PROGRAM pouStationUnits
VAR
	row1: FB_HMI_Control;
	row2: FB_HMI_Control;
	row3: FB_HMI_Control;
	row4: FB_HMI_Control;
	row5: FB_HMI_Control;
	row6: FB_HMI_Control;
	row7: FB_HMI_Control;
	row8: FB_HMI_Control;
	row9: FB_HMI_Control;
	row10: FB_HMI_Control;
	tNumberOfPages: REAL;
	tCalcNumberOfPages: REAL;
	row11: FB_HMI_Control;
	row12: FB_HMI_Control;
	row13: FB_HMI_Control;
	row14: FB_HMI_Control;
	row15: FB_HMI_Control;
	row16: FB_HMI_Control;
	row17: FB_HMI_Control;
	row18: FB_HMI_Control;
	row19: FB_HMI_Control;
	row20: FB_HMI_Control;
	row21: FB_HMI_Control;
	row22: FB_HMI_Control;
	row23: FB_HMI_Control;
	row24: FB_HMI_Control;
	//StationNativeMotionRows: ARRAY[0..99] OF typeMotionRow;
	ceil: LREAL;
END_VAR

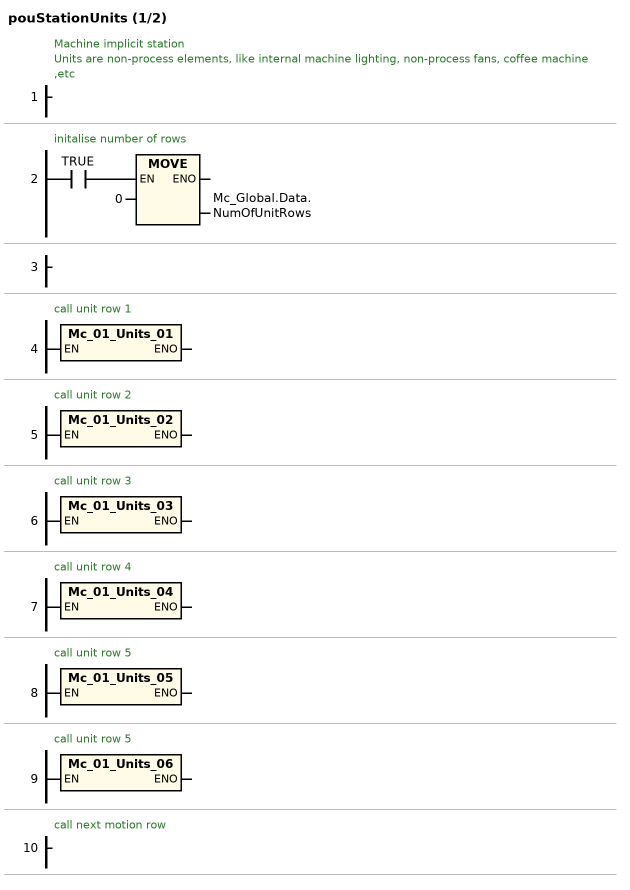
// NETWORK 1
// Machine implicit station
// Units are non-process elements, like internal machine lighting, non-process fans, coffee machine ,etc

// NETWORK 2
// initalise number of rows
Mc_Global.Data.NumOfUnitRows := 0;

// NETWORK 3

// NETWORK 4
// call unit row 1
Mc_01_Units_01();

// NETWORK 5
// call unit row 2
Mc_01_Units_02();

// NETWORK 6
// call unit row 3
Mc_01_Units_03();

// NETWORK 7
// call unit row 4
Mc_01_Units_04();

// NETWORK 8
// call unit row 5
Mc_01_Units_05();

// NETWORK 9
// call unit row 5
Mc_01_Units_06();

// NETWORK 10
// call next motion row

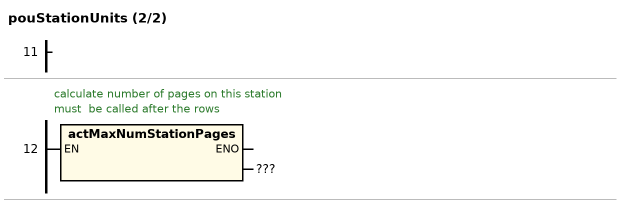
// NETWORK 11

// NETWORK 12
// calculate number of pages on this station
// must  be called after the rows
actMaxNumStationPages();

ACTION actMaxNumStationPages:
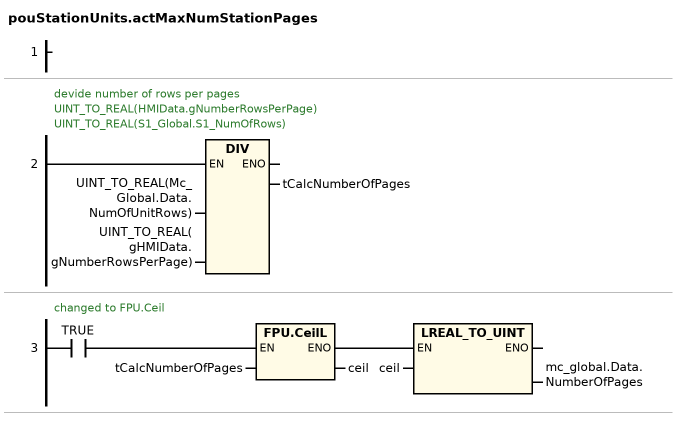
// NETWORK 1

// NETWORK 2
// devide number of rows per pages
// UINT_TO_REAL(HMIData.gNumberRowsPerPage)
// UINT_TO_REAL(S1_Global.S1_NumOfRows)
tCalcNumberOfPages := (UINT_TO_REAL(Mc_Global.Data.NumOfUnitRows)) / (UINT_TO_REAL(gHMIData.gNumberRowsPerPage));

// NETWORK 3
// changed to FPU.Ceil
ceil := FPU.CeilL(tCalcNumberOfPages);
mc_global.Data.NumberOfPages := LREAL_TO_UINT(ceil);
END_ACTION

END_PROGRAM

(* stored: Version 1.1.0.1, ProductVersion 3.1.4024.12
   POU pouStationUnits: Id {73b32ded-9dff-42ce-81b2-f5e2a8400972}, SpecialFunc None
   Action actMaxNumStationPages: Id {a6ae48a4-2f66-4d35-9de1-b2d5d7451ce0} *)
